PROGRAM MAIN
VAR
    CycleTimer : TON;
END_VAR

CycleTimer(IN := NOT CycleTimer.Q, PT := T#1S);

IF CycleTimer.Q THEN
    MachineData.PartCount := MachineData.PartCount + 1;
    MachineData.MotorTemp       := MachineData.MotorTemp + 0.1;
    MachineData.ConveyorRunning := TRUE;
END_IF

END_PROGRAM

(* stored: Version 1.1.0.1, ProductVersion 3.1.4026.18
   POU MAIN: Id {c7a1bc91-dcde-41b5-a4ba-f34c52173b03}, SpecialFunc None *)
